(* PLC project DemoProject *)

TYPE MotorType : STRUCT
  Running : BOOL;
  Rpm : INT := 1500;
END_STRUCT;
END_TYPE

PROGRAM Main
  VAR
    Count : DINT := 7;
  END_VAR

Count := Count + 1;
END_PROGRAM

PROGRAM Rung1

(* LD diagram, written out as Structured Text *)
Motor := Start;
END_PROGRAM

CONFIGURATION Config
  RESOURCE Res ON PLC
    VAR_GLOBAL
      Temp_PV : REAL := 20.0;
      Enable : BOOL := TRUE;
      Retained : LREAL;
    END_VAR
  END_RESOURCE
END_CONFIGURATION
